SUBAPPLICATION Uebung_093b (* Beispiel für E_N_TABLE *)
  (* Standard: 61499-2; Description: Copyright (c) 2023 Meisterschulen am Ostbahnhof This program and the accompanying materials are made available under the terms of the Eclipse Public License 2.0 which is available at https://www.eclipse.org/legal/epl-2.0/ SPDX-License-Identifier: EPL-2.0 *)
  (* Version 1.0, 2023-10-23, Franz Höpfinger, Meisterschulen am Ostbahnhof *)
  IMPORT logiBUS::io::DI::logiBUS_DI;
  IMPORT logiBUS::io::DI::logiBUS_DI_Events;
  IMPORT logiBUS::io::DQ::logiBUS_DO;
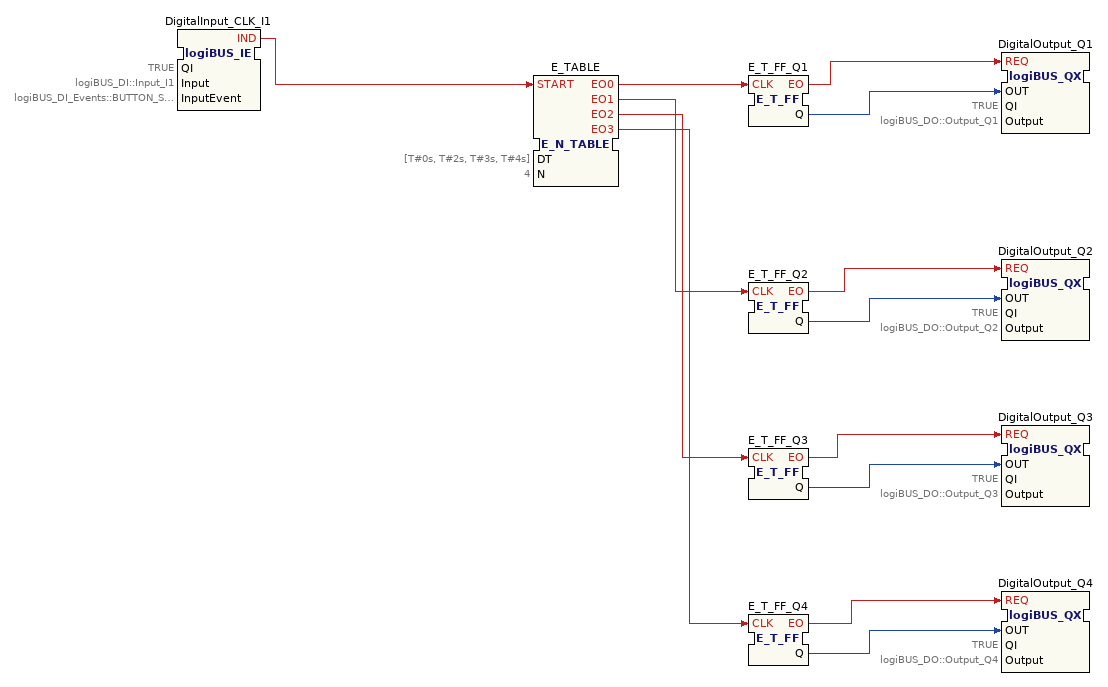
  (* E_TABLE wird 4 Events ausgeben, das erste sofort nach dem Click, das letzte 9s nach dem Click [T#0s, T#2s, T#3s, T#4s] *)
  FBS
    E_TABLE : iec61499::events::E_N_TABLE(DT := [T#0s, T#2s, T#3s, T#4s], N := 4);
    DigitalInput_CLK_I1 : logiBUS::io::DI::logiBUS_IE(QI := TRUE, Input := logiBUS_DI::Input_I1, InputEvent := logiBUS_DI_Events::BUTTON_SINGLE_CLICK);
    E_T_FF_Q2 : iec61499::events::E_T_FF;
    E_T_FF_Q4 : iec61499::events::E_T_FF;
    DigitalOutput_Q1 : logiBUS::io::DQ::logiBUS_QX(QI := TRUE, Output := logiBUS_DO::Output_Q1);
    E_T_FF_Q3 : iec61499::events::E_T_FF;
    DigitalOutput_Q3 : logiBUS::io::DQ::logiBUS_QX(QI := TRUE, Output := logiBUS_DO::Output_Q3);
    E_T_FF_Q1 : iec61499::events::E_T_FF;
    DigitalOutput_Q2 : logiBUS::io::DQ::logiBUS_QX(QI := TRUE, Output := logiBUS_DO::Output_Q2);
    DigitalOutput_Q4 : logiBUS::io::DQ::logiBUS_QX(QI := TRUE, Output := logiBUS_DO::Output_Q4);
  END_FBS
  EVENT_CONNECTIONS
    DigitalInput_CLK_I1.IND TO E_TABLE.START;
    E_T_FF_Q1.EO TO DigitalOutput_Q1.REQ;
    E_T_FF_Q3.EO TO DigitalOutput_Q3.REQ;
    E_T_FF_Q2.EO TO DigitalOutput_Q2.REQ;
    E_T_FF_Q4.EO TO DigitalOutput_Q4.REQ;
    E_TABLE.EO0 TO E_T_FF_Q1.CLK;
    E_TABLE.EO1 TO E_T_FF_Q2.CLK;
    E_TABLE.EO2 TO E_T_FF_Q3.CLK;
    E_TABLE.EO3 TO E_T_FF_Q4.CLK;
  END_CONNECTIONS
  DATA_CONNECTIONS
    E_T_FF_Q1.Q TO DigitalOutput_Q1.OUT;
    E_T_FF_Q4.Q TO DigitalOutput_Q4.OUT;
    E_T_FF_Q2.Q TO DigitalOutput_Q2.OUT;
    E_T_FF_Q3.Q TO DigitalOutput_Q3.OUT;
  END_CONNECTIONS
END_SUBAPPLICATION
